Universal Robots PolyScope program: DoneRoboProg.urp

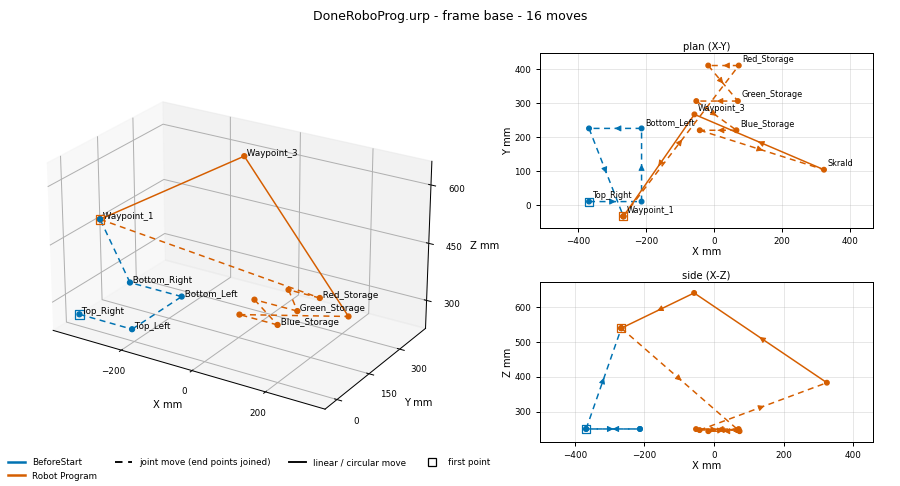
[picture p0: tool path of DoneRoboProg.urp in frame base, 16 of 17 moves have a stored position in this frame; points joined in program order, loops and branches not executed]
Program DoneRoboProg (installation=default directory=/programs/usbdisk_1 createdIn=3.9.1.64192 lastSavedIn=3.9.1.64192 robotSerialNumber=2016331617)
Calibrated DH parameters: a=[-0.000045, -0.22956, -0.153032, 0.000019, 0.0001, 0]; d=[0.152163, -856.35044, 904.692211, -48.229373, 0.085425, 0.082565]; alpha=[1.571202, -0.000097, 0.003084, 1.571016, -1.571253, 0]; deltaTheta=[-0.00003, 0.346154, 0.426056, -0.772366, 0.00006, 0.000029]
BeforeStart
  Loop Counting (count=2) loopVariable(name=Loop_2)
    MoveJ speed 60 deg/s, acceleration 80 deg/s^2 (useActiveTCP=true)
      Waypoint Top_Right: TCP in base x=-367.597 y=10.283 z=250.202 mm, rx=3.0998 ry=-0.0003 rz=0.0005 rad; joints [-19.998, -76.118, 91.028, -104.096, -87.648, 70.138] deg
      Wait Sleep waitTime=2
      Waypoint Top_Left: TCP in base x=-212.881 y=10.267 z=250.174 mm, rx=3.0998 ry=-0.0002 rz=0.0007 rad; joints [-35.605, -118.18, 126.872, -97.298, -87.938, 54.508] deg
      Wait Sleep waitTime=2
      Waypoint Bottom_Left: TCP in base x=-212.851 y=225.763 z=250.159 mm, rx=3.0998 ry=-0.0004 rz=0.0008 rad; joints [-68.254, -89.612, 105.936, -104.107, -89.029, 21.884] deg
      Wait Sleep waitTime=2
      Waypoint Bottom_Right: TCP in base x=-367.577 y=225.743 z=250.179 mm, rx=3.0999 ry=-0.0003 rz=0.0006 rad; joints [-47.033, -60.178, 67.814, -95.891, -88.259, 43.078] deg
      Wait Sleep waitTime=2
  Loop Forever
    Script: conres = socket_open("192.168.137.1",23)
    Script: textmsg(conres)
    If conres ≟  True
      Script: break
  Script: targetPos=p[0, 0, 0, 0, 0, 0]
  Script: receiveFromServ=[0, 0, 0, 0, 0, 0, 0, 0]
  MoveJ speed 60 deg/s, acceleration 80 deg/s^2 (useActiveTCP=true)
    Waypoint Waypoint_1: TCP in base x=-266.42 y=-33.236 z=539.766 mm, rx=-1.5425 ry=0.3637 rz=0.4165 rad; joints [0.597, -76.494, 58.72, -159.143, -178.731, 31.561] deg
  Script: Kalibrer="Kalibrering"
  Script: socket_send_string(Kalibrer)
  Loop While (checkContinuously=false) expression=conres≟ True
    Script: KaliSlut=socket_read_ascii_float(1)
    Script: textmsg(KaliSlut)
    If KaliSlut[1]≟100
      Script: break
Robot Program (runOnlyOnce=false)
  Set DigitalOutput pin=tool_out[0]; digitalValue=0
  MoveJ speed 60 deg/s, acceleration 80 deg/s^2 (useActiveTCP=true)
    Waypoint Waypoint_1: TCP in base x=-266.42 y=-33.236 z=539.766 mm, rx=-1.5425 ry=0.3637 rz=0.4165 rad; joints [0.597, -76.494, 58.72, -159.143, -178.731, 31.561] deg
  Script: sendToServer="Klar"
  Script: socket_send_string(sendToServer)
  Loop While (checkContinuously=false) expression=conres≟ True
    Script: receiveFromServ=socket_read_ascii_float(7)
    Script: textmsg(receiveFromServ)
    If receiveFromServ[7]≟1
      Script: break
    ElseIf receiveFromServ[7]≟2
      Script: break
    ElseIf receiveFromServ[7]≟3
      Script: break
    ElseIf receiveFromServ[7]≟4
      Script: break
  Loop Forever
    Script: targetPos=p[receiveFromServ[1],receiveFromServ[2],receiveFromServ[3],receiveFromServ[4],receiveFromServ[5],receiveFromServ[6]]
    Script: textmsg(targetPos)
    If targetPos≠p[0, 0, 0, 0, 0, 0]
      MoveL speed 250 mm/s, acceleration 1200 mm/s^2 (useActiveTCP=true) feature=Base
        Waypoint Waypoint (Variable): variable=targetPos
      Script: break
  Set ExpressionOutput pin=tool_out[0]; expression=True
  Wait Sleep waitTime=2
  MoveJ speed 60 deg/s, acceleration 80 deg/s^2 (useActiveTCP=true)
    Waypoint Waypoint_1: TCP in base x=-266.42 y=-33.236 z=539.766 mm, rx=-1.5425 ry=0.3637 rz=0.4165 rad; joints [0.597, -76.494, 58.72, -159.143, -178.731, 31.561] deg
  Wait Sleep waitTime=2
  If receiveFromServ[7]≟1
    If Red≟0
      MoveJ speed 60 deg/s, acceleration 80 deg/s^2 (useActiveTCP=true)
        Waypoint Red_Storage: TCP in base x=73.399 y=410.879 z=243.753 mm, rx=-2.6828 ry=-1.565 rz=0.0637 rad; joints [-116.419, -63.852, 75.621, -100.933, -86.913, -86.822] deg
        Set ExpressionOutput pin=tool_out[0]; expression=False
        Wait Sleep waitTime=1
        Set IncrementVariable installationVariable=Red
    ElseIf Red≠0
      MoveJ speed 60 deg/s, acceleration 80 deg/s^2 (useActiveTCP=true)
        Waypoint Red_Storage_2: TCP in base x=-16.551 y=410.893 z=243.78 mm, rx=-2.6827 ry=-1.5649 rz=0.0635 rad; joints [-104.259, -65.548, 78.427, -102.698, -86.806, -74.639] deg
        Set ExpressionOutput pin=tool_out[0]; expression=False
        Wait Sleep waitTime=1
  ElseIf receiveFromServ[7]≟2
    If Green≟0
      MoveJ speed 60 deg/s, acceleration 80 deg/s^2 (useActiveTCP=true)
        Waypoint Green_Storage: TCP in base x=70.718 y=306.264 z=249.848 mm, rx=-2.7016 ry=-1.4787 rz=0.0435 rad; joints [-125.132, -89.524, 106.948, -107.552, -86.025, -92.369] deg
        Set ExpressionOutput pin=tool_out[0]; expression=False
        Wait Sleep waitTime=1
        Set IncrementVariable installationVariable=Green
    ElseIf Green≠0
      MoveJ speed 60 deg/s, acceleration 80 deg/s^2 (useActiveTCP=true)
        Waypoint Green_Storage_2: TCP in base x=-51.686 y=306.259 z=249.829 mm, rx=-2.7018 ry=-1.4787 rz=0.0435 rad; joints [-102.735, -90.747, 108.788, -109.634, -86.367, -69.922] deg
        Set ExpressionOutput pin=tool_out[0]; expression=False
        Wait Sleep waitTime=1
  ElseIf receiveFromServ[7]≟3
    If Blue≟0
      MoveJ speed 60 deg/s, acceleration 80 deg/s^2 (useActiveTCP=true)
        Waypoint Blue_Storage: TCP in base x=66.478 y=220.285 z=246.895 mm, rx=-2.7077 ry=-1.5077 rz=0.0571 rad; joints [-137.325, -112.52, 124.913, -100.928, -87.046, -105.446] deg
        Set ExpressionOutput pin=tool_out[0]; expression=False
        Wait Sleep waitTime=1
        Set IncrementVariable installationVariable=Blue
    ElseIf Blue≠0
      MoveJ speed 60 deg/s, acceleration 80 deg/s^2 (useActiveTCP=true)
        Waypoint Blue_Storage_2: TCP in base x=-41.487 y=220.272 z=246.895 mm, rx=-2.7076 ry=-1.5078 rz=0.0571 rad; joints [-110.926, -115.037, 126.823, -101.738, -86.682, -79.016] deg
        Set ExpressionOutput pin=tool_out[0]; expression=False
        Wait Sleep waitTime=1
  ElseIf receiveFromServ[7]≟4
    MoveJ speed 60 deg/s, acceleration 80 deg/s^2 (useActiveTCP=true)
      Waypoint Skrald: TCP in base x=324.295 y=104.113 z=383.107 mm, rx=-2.9845 ry=-0.398 rz=-0.2817 rad; joints [-183.781, -86.97, 72.213, -84.486, -81.166, -108.163] deg
      Set ExpressionOutput pin=tool_out[0]; expression=False
      Wait Sleep waitTime=1
  Wait Sleep waitTime=1
  Script: targetPos=p[0, 0, 0, 0, 0, 0]
  MoveL speed 250 mm/s, acceleration 1200 mm/s^2 (useActiveTCP=true) feature=Base
    Waypoint Waypoint_3: TCP in base x=-57.227 y=267.03 z=641.08 mm, rx=-1.4722 ry=-0.7316 rz=-0.9403 rad; joints [-214.721, -128.931, 35.953, -85.767, 26.68, -62.197] deg
    Waypoint Waypoint_1: TCP in base x=-266.42 y=-33.236 z=539.766 mm, rx=-1.5425 ry=0.3637 rz=0.4165 rad; joints [0.597, -76.494, 58.72, -159.143, -178.731, 31.561] deg
